FUNCTION_BLOCK FB_LoadingStation IMPLEMENTS I_WorkingStation
VAR_INPUT
END_VAR
VAR_OUTPUT
END_VAR
VAR
END_VAR

PROPERTY prTableInPosition : BOOL
GET
END_GET
SET
END_SET
END_PROPERTY

{warning 'add property implementation'}
PROPERTY prTableRotationInterlock : BOOL
GET
END_GET
SET
END_SET
END_PROPERTY

{warning 'add property implementation'}
PROPERTY prTableRotationRequest : BOOL
GET
END_GET
SET
END_SET
END_PROPERTY

END_FUNCTION_BLOCK

(* stored: Version 1.1.0.1, ProductVersion 3.1.4024.15
   POU FB_LoadingStation: Id {0739b0e9-6a0b-43e8-b760-d31010e6020e}, SpecialFunc None
   Property prTableInPosition: Id {592cf85c-3254-4812-b020-5d141833f6ab}
   Get Get: Id {217c66a4-f5be-4f35-b16e-a6b86af79b22}
   Set Set: Id {bb7ede60-fba5-4c19-8c00-ebcefea92104}
   Property prTableRotationInterlock: Id {e5fc254a-5609-4be3-84a7-f8c244dac0b1}
   Get Get: Id {b7a6cd8a-205a-4ef0-80ee-061e503f9f54}
   Set Set: Id {dd4a82e4-3071-4331-955b-6cba30b3edf6}
   Property prTableRotationRequest: Id {4f6b0926-f186-40fb-a73a-e615918a2a53}
   Get Get: Id {e1c3145f-d20b-41e6-89c1-66bdfe48409e}
   Set Set: Id {cd771a07-006e-4e10-81db-f4cea774d852} *)
